TYPE ST_OutputsFastDoor :
STRUCT
	HW		: ST_HW_OutputsFastDoor; //Hardware output
END_STRUCT
END_TYPE

(* stored: Version 1.1.0.1, ProductVersion 3.1.4024.9
   DUT ST_OutputsFastDoor: Id {2cafb99a-1b2d-4a56-981a-111ae9e78de9} *)
